PROGRAM MAIN
VAR
	fbTCP_IP_Server: FB_TCP_IP_Server;
	fbTCP_IP_ServerClientConnection: FB_TCP_IP_ServerClientConnection;
END_VAR
VAR CONSTANT
END_VAR


fbTCP_IP_Server(
	sSrvNetId:= , 
	sLocalHost:= , 
	nLocalPort:= , 
	bListen:= , 
	bClose:= , 
	bReset:= , 
	TIMEOUT:= );

fbTCP_IP_ServerClientConnection();

END_PROGRAM

(* stored: Version 1.1.0.1, ProductVersion 3.1.4024.13
   POU MAIN: Id {90fa3c98-d7c6-42f6-8b49-07c136b3c71a}, SpecialFunc None *)
